{attribute 'qualified_only'}
VAR_GLOBAL
	
END_VAR

(* stored: Version 1.1.0.1, ProductVersion 3.1.4024.9
   GVL GVL: Id {c5512198-46ab-4fa2-b20b-019005d511ba} *)
